PROGRAM P1_Camera
VAR
		stPos					:ST_PosData;
		tCycleTime				:TON;
		i						:INT;
		tPalletStartTime		:TON;
		nCycle_Idx				:BYTE;
		arrMES_Temp				:ARRAY [0..2] OF ST_P1MesData;
END_VAR

(*Időzítők***************************************************)
IF (stPos.nState>10000) AND (stPos.nState<100000) AND NOT tCycleTime.Q THEN
	stPos.nCycleTime := TIME_TO_REAL(tCycleTime.ET)/1000;
END_IF
tCycleTime(IN:= (stPos.nState>10000) AND (stPos.nState<150000), PT:= T#200S);							// A palettára várakozás nincs beszámolva
tPalletStartTime(IN:= NOT i_bP2PalletSensor AND fbConveyor_1.bMotorOn, PT:= T#4S);					// Alaphelyzet felvétel késleltetése!

(*Triggerek**************************************************)

(*Vész rendszer**********************************************)
IF	(NOT (i_bEmyOK AND fbDoor.bDoorsLocked) AND stPos.nState > 0) OR									// Nincs vészkör, vagy
	(NOT i_bDoorOK AND (stPos.nState>=60 AND stPos.nState<=1000)) OR									// alaphelyzetfelvétel közbe megszűnik az ajtókör vagy
	(NOT i_bDoorOK AND (stPos.nState>=10060 AND stPos.nState<=100060)) THEN							// folyamat közbe megszűnik az ajtókör 
		stPos.nState := 0;
END_IF;

(*Hibakezelés************************************************)
IF stPos.nState > 0 AND stPos.nState < 150000 THEN
	stPos.nStateLast := stPos.nState;
	IF	fbP1Lift.bError OR
		fbP1PalletDataExchange.bError OR
		(fbP1AxisX.bError AND i_bDoorOK (*AND stP1.nState >= 500*)) OR
		(fbP1AxisY.bError AND i_bDoorOK (*AND stP1.nState >= 500*)) OR
		(fbP1AxisZ.bError AND i_bDoorOK (*AND stP1.nState >= 500*)) OR
		stPos.bError THEN
			stPos.nState := 200000;
	END_IF
END_IF

(*Engedélyek *************************************************)
IF stPos.nState <= 10000
	OR stPos.nState = 100000
	OR stPos.nState = 150000
	OR stPos.nState >= 200000
THEN
	stPos.bManualModeEnable := TRUE;
ELSE
	stPos.bManualModeEnable := FALSE;
END_IF

IF stPos.nState = 0
	OR stPos.nState = 10000
	OR stPos.nState = 100000
	OR stPos.nState = 150000
	OR stPos.nState >= 200000
THEN
	stPos.bDoorOpenEnable := TRUE;
ELSE
	stPos.bDoorOpenEnable := FALSE;
END_IF

(*Kézi üzem *************************************************)
IF bManualMode THEN
	stPos.nState := 150000;
END_IF

(*Automata üzem *********************************************)
CASE stPos.nState OF
{region "Init process"}
	0:		stPos.sState := CONCAT(UDINT_TO_STRING(stPos.nState) ,' - Vészkör vagy ajtókör bontva - Működtetések törlése');
			fbP1AxisX.bGoPosition := FALSE;
			fbP1AxisY.bGoPosition := FALSE;
			fbP1AxisZ.bGoPosition := FALSE;
			fbP1Lift.bBasePosCmd := TRUE;
			fbP1Lift.bWorkPosCmd := FALSE;
			fbP1PalletDataExchange.eCommand := NoCmd;
			stPos.bError := FALSE;
			stPos.nErrorCode := 0;
			IF i_bDoorOK THEN
				IF bStepEnable THEN
					stPos.nState := stPos.nState + 20;
				END_IF
			END_IF
			
	20:		stPos.sState := CONCAT(UDINT_TO_STRING(stPos.nState) ,' - Alaphelyzetfelvétel - Kiemelő alaphelyzetbe');
			fbP1Lift.bBasePosCmd := TRUE;
			fbP1Lift.bWorkPosCmd := FALSE;
			IF fbP1Lift.bBasePosStab THEN
				IF bStepEnable THEN
					stPos.nState := stPos.nState + 20;
				END_IF
			END_IF
			
	40:		stPos.sState := CONCAT(UDINT_TO_STRING(stPos.nState) ,' - AX5805 safety ellenőrzés');	
			IF (i_bAX5805ErrorX OR i_bAX5805ErrorX) AND NOT q_bAX5805_Ack THEN
				q_bAX5805_Ack := TRUE;
			ELSIF NOT (i_bAX5805ErrorX OR i_bAX5805ErrorY OR i_bAX5805ErrorZ) THEN
				q_bAX5805_Ack := FALSE;
				IF bStepEnable THEN
					stPos.nState := stPos.nState + 20;
				END_IF
			END_IF

	60:		stPos.sState := CONCAT(UDINT_TO_STRING(stPos.nState) ,' - Szervo X tengely drive ellenőrzés');	
			IF NOT fbP1AxisX.Axis.Status.DriveDeviceError THEN
				IF bStepEnable THEN
					stPos.nState := stPos.nState + 20;
				END_IF
			END_IF

	80:		stPos.sState := CONCAT(UDINT_TO_STRING(stPos.nState) ,' - Szervo X tengely NC ellenőrzés');	
			IF NOT fbP1AxisX.Axis.Status.Error THEN
				IF bStepEnable THEN
					stPos.nState := stPos.nState + 20;
				END_IF
			END_IF

	100:	stPos.sState := CONCAT(UDINT_TO_STRING(stPos.nState) ,' - Szervo X tengely ellenőrzés');	
			IF fbP1AxisX.nState = 1000 THEN
				IF bStepEnable THEN
					stPos.nState := stPos.nState + 20;
				END_IF
			END_IF
			
	120:	stPos.sState := CONCAT(UDINT_TO_STRING(stPos.nState) ,' - Szervo Y tengely drive ellenőrzés');	
			IF NOT fbP1AxisY.Axis.Status.DriveDeviceError THEN
				IF bStepEnable THEN
					stPos.nState := stPos.nState + 20;
				END_IF
			END_IF

	140:	stPos.sState := CONCAT(UDINT_TO_STRING(stPos.nState) ,' - Szervo Y tengely NC ellenőrzés');	
			IF NOT fbP1AxisY.Axis.Status.Error THEN
				IF bStepEnable THEN
					stPos.nState := stPos.nState + 20;
				END_IF
			END_IF

	160:	stPos.sState := CONCAT(UDINT_TO_STRING(stPos.nState) ,' - Szervo Y tengely ellenőrzés');	
			IF fbP1AxisY.nState = 1000 THEN
				IF bStepEnable THEN
					stPos.nState := stPos.nState + 20;
				END_IF
			END_IF

	180:	stPos.sState := CONCAT(UDINT_TO_STRING(stPos.nState) ,' - Szervo Z tengely drive ellenőrzés');	
			IF NOT fbP1AxisZ.Axis.Status.DriveDeviceError THEN
				IF bStepEnable THEN
					stPos.nState := stPos.nState + 20;
				END_IF
			END_IF

	200:	stPos.sState := CONCAT(UDINT_TO_STRING(stPos.nState) ,' - Szervo Z tengely NC ellenőrzés');	
			IF NOT fbP1AxisZ.Axis.Status.Error THEN
				IF bStepEnable THEN
					stPos.nState := stPos.nState + 20;
				END_IF
			END_IF

	220:	stPos.sState := CONCAT(UDINT_TO_STRING(stPos.nState) ,' - Szervo Z tengely ellenőrzés');	
			IF fbP1AxisZ.nState = 1000 THEN
				IF bStepEnable THEN
					stPos.nState := 500;
				END_IF
			END_IF
	 
			
	500:	stPos.sState := CONCAT(UDINT_TO_STRING(stPos.nState) ,' - Z tengely alaphelyzetbe mozgatása');			
			fbP1AxisZ.rPosition1 := 0;
			fbP1AxisZ.rVelocity1 := 100;
			fbP1AxisZ.bGoPosition := TRUE;
			IF fbP1AxisZ.bDone THEN
				IF bStepEnable THEN
					fbP1AxisZ.bGoPosition := FALSE;
					stPos.nState := stPos.nState + 20;
				END_IF
			END_IF
			
	520:	stPos.sState := CONCAT(UDINT_TO_STRING(stPos.nState) ,' - X tengely alaphelyzetbe mozgatása');			
			fbP1AxisX.rPosition1 := 0;
			fbP1AxisX.rVelocity1 := 100;
			fbP1AxisX.bGoPosition := TRUE;
			IF fbP1AxisX.bDone THEN
				IF bStepEnable THEN
					fbP1AxisX.bGoPosition := FALSE;
					stPos.nState := stPos.nState + 20;
				END_IF
			END_IF
			
	540:	stPos.sState := CONCAT(UDINT_TO_STRING(stPos.nState) ,' - Y tengely alaphelyzetbe mozgatása');			
			fbP1AxisY.rPosition1 := 0;
			fbP1AxisY.rVelocity1 := 100;
			fbP1AxisY.bGoPosition := TRUE;
			IF fbP1AxisY.bDone THEN
				IF bStepEnable THEN
					fbP1AxisY.bGoPosition := FALSE;
					stPos.nState := stPos.nState + 20;
				END_IF
			END_IF
					 
	560:	stPos.sState := CONCAT(UDINT_TO_STRING(stPos.nState) ,' - Várakozás paletta mozgásra a pzíciók között');
			IF tPalletStartTime.Q THEN									// Normál esetben nem kerülhet ebbe az állapotba a berendezés!
				IF bStepEnable THEN										// Ha viszont P1 elengedi a palettát, amin jó termék van, és az még nem érkezik meg P2-be
					stPos.nState := 10000;								// a következő paletta ami üres megérkezik P1-be, ekkor nyomnak egy vészstopot, kinyitják az ajtót és visszahúzzák
				END_IF													// a palettát P2 elől, akkor induláskor P1 rögtön elengedné az üres palettát igy P2-be 2 paletta érkezne!!!!
			END_IF														// Ebből a hibából automatikusan csak selejtezéssel lehetne kiszedni az állomást!!! Ez nem lenne túl szerencsés!!

{endregion}
			
(* Alaphelyzet *********************************************************************)
	10000:	stPos.sState := CONCAT(UDINT_TO_STRING(stPos.nState) ,' - Alaphelyzet, termékre vár');
			IF fbP1RFID.bTagPresent AND fbP1Stopper.bPalletAtStopper AND NOT bP1ScrapRepeatError THEN
				IF bStepEnable THEN
					stPos.nState := stPos.nState + 20;
				END_IF
			END_IF	

{region "Pallet receive"}
	(*-----=== Hordozólap adatok lekérdezése ST10-től ===-----*)
	10020:	stPos.sState := CONCAT(UDINT_TO_STRING(stPos.nState) ,' - Paletta adatok lekérdezése');
			fbP1PalletDataExchange.nIndex := fbP1RFID.nTAGData;
			IF bStepEnable THEN
				fbP1PalletDataExchange.eCommand := Read;
				stPos.nState := stPos.nState + 20;
			END_IF
			
	(*-----=== Hordozólap adatok lekérdezése ST10-től ===-----*)
	10040:	stPos.sState := CONCAT(UDINT_TO_STRING(stPos.nState) ,' - Paletta adatok lekérdezése');
			IF fbP1PalletDataExchange.bDone AND NOT fbP1PalletDataExchange.bError THEN
				IF bStepEnable THEN
					fbP1PalletDataExchange.eCommand := NoCmd;
					stPos.nState := stPos.nState + 20;
				END_IF
			END_IF

	(*-----=== Hordozólap adatok kiértékelése ===-----*)
	10060:	stPos.sState := CONCAT(UDINT_TO_STRING(stPos.nState) ,' - Paletta adatok lekérdezése');
			IF		stP1PalletData.nPalletState = 2 AND			// OK termék a palettán
					stP1PalletData.nDone.3 AND					// Diszpenzálás kész
					NOT stP1PalletData.nDone.4 THEN				// Kamerás ell. még nincs kész
						IF bStepEnable THEN						// Mehet a kiemelés -> Normál folyamat
							nCycle_Idx := 0;

							arrMES_Temp[0].nOP_Index := nP1GapFillerCheckCover_Index;
							arrMES_Temp[0].sDMC_Code := stP1PalletData.sCoverCode;
							arrMES_Temp[0].sOP_Name := 'OP_GAP_FILLER_CHK_COVER';
							
							arrMES_Temp[1].nOP_Index := nP1CheckSim_Index;
							arrMES_Temp[1].sDMC_Code := stP1PalletData.sMRTCode;
							arrMES_Temp[1].sOP_Name := 'OP_CHECK_SIM';
	
							arrMES_Temp[2].nOP_Index := nP1CheckComponent_Index;
							arrMES_Temp[2].sDMC_Code := stP1PalletData.sMRTCode;
							arrMES_Temp[2].sOP_Name := 'OP_CHECK_COMPONENT';
	
							stPos.nState := stPos.nState + 20;
						END_IF
			ELSIF	stP1PalletData.nPalletState = 41 THEN		// Teszt hordozólap a kamerához
						IF bStepEnable THEN						// Még nincs funkció -> Tovább engedés
							stPos.nState := 96060; //????
						END_IF
			ELSIF	stP1PalletData.nPalletState = 2 AND			// OK termék a palettán
					NOT stP1PalletData.nDone.3 THEN				// Diszpenzálás nincs kész !
						IF bStepEnable THEN						// Átemelt hordozólap!?!? -> Selejtezés
							stP1PalletData.nPalletState := 1;
							stP1PalletData.nDone.4	:= TRUE;
							stP1PalletData.nErrorCode := 4100;
							stPos.nState := 96000;
						END_IF
			ELSIF	stP1PalletData.nPalletState = 1 THEN		// Selejt termék a palettán
						IF bStepEnable THEN						// Nincs kiemelés -> Tovább engedés
							stPos.nState := 96060;
						END_IF
			ELSIF	stP1PalletData.nPalletState = 0 THEN		// Üres paletta
						IF bStepEnable THEN						// Nincs kiemelés -> Tovább engedés
							stPos.nState := 96060;
						END_IF
			ELSE												// Nincs teendő, más állomásnak szánt hordozólap
						IF bStepEnable THEN						// Nincs kiemelés -> Tovább engedés
							stPos.nState := 96060;
						END_IF			
			END_IF

	(*-----=== MES engedély ellenőrzése ===-----*)
	10080:	stPos.sState := CONCAT(UDINT_TO_STRING(stPos.nState) ,' - MES engedély ellenőrzése');
			IF bMesEnable THEN
				IF bStepEnable THEN
					stPos.nState := 14000;
				END_IF
			ELSE
				IF bStepEnable THEN
					stPos.nState := 16000;
				END_IF				
			END_IF
{endregion}

{region "Normal process"} 
(*-----=== Recept lista kezelés ===-----*)
(* Get MRT OP state *)
14000:		stPos.sState := CONCAT(UDINT_TO_STRING(stPos.nState) ,' - Get OP state MRT (1026)');
			IF fbP1MesInterface.GET_CURRENT_OPERATION_STATE(stP1PalletData.sMRTCode, 0,stP1MesOpState) THEN
				IF stP1MesResp.RESP_CODE = '0' or stP1MesResp.RESP_CODE = '377'	THEN									// MRT OP state OK
					IF bStepEnable THEN
						stP1MrtMaterial.MATERIAL := stP1MesOpState.MAT_NO;
						stP1MrtMaterial.REVISION := stP1MesOpState.REVISION;
						nCycle_Idx := 0;
						stPos.nState := 14100;
					END_IF		
				ELSE
					IF bStepEnable THEN													// Get OP state hiba
						stP1PalletData.nPalletState := 1;
						stP1PalletData.nDone.4	:= TRUE;
							stP1PalletData.nErrorCode := 4101;
						stPos.nState := 96000;
					END_IF
				END_IF
			END_IF

	 
14100:		stPos.sState := CONCAT(UDINT_TO_STRING(stPos.nState) ,' - Get Material Custom Data (1037)');
			IF fbP1MesInterface.GET_MAT_CUSTOM_DATA(stP1MrtMaterial, 0) THEN
				IF stP1MesResp.RESP_CODE = '0'	THEN									// Get Custom Data OK
					IF bStepEnable THEN
						stPos.nState := stPos.nState + 20;
					END_IF		
				ELSE
					IF bStepEnable THEN													// Get Custom Data hiba
						stP1PalletData.nPalletState := 1;
						stP1PalletData.nDone.4	:= TRUE;
							stP1PalletData.nErrorCode := (4102 + nCycle_Idx);
						stPos.nState := 96000;
					END_IF
				END_IF
			END_IF		  

14120:		stPos.sState := CONCAT(UDINT_TO_STRING(stPos.nState) ,' - Get Custom Data By Key');
			IF fbP1MesInterface.GET_CUSTOM_DATA_BY_KEY(CONCAT(arrMES_Temp[nCycle_Idx].sOP_Name, '_R'), arrMES_Temp[nCycle_Idx].sOP_CustomData) THEN
				IF arrMES_Temp[nCycle_Idx].sOP_CustomData <> ''	THEN					// Get Custom Data by key OK
					IF bStepEnable THEN
						arrMES_Temp[nCycle_Idx].sOP_ReceipeList := arrMES_Temp[nCycle_Idx].sOP_CustomData;
						stPos.nState := stPos.nState + 20;
					END_IF		
				ELSE
					IF bStepEnable THEN													// Get Custom Data by key hiba
						stP1PalletData.nPalletState := 1;
						stP1PalletData.nDone.4	:= TRUE;
							stP1PalletData.nErrorCode := (4103 + nCycle_Idx);
						stPos.nState := 96000;
					END_IF
				END_IF
			END_IF		  

14140:		stPos.sState := CONCAT(UDINT_TO_STRING(stPos.nState) ,' - Recept lista ellenőrzése');   
			IF nCycle_Idx >= 2 THEN
				IF bStepEnable THEN						// Custom fied-ek átemelve -> Gyí, gyí gyí !!!
					nCycle_Idx := 0;
					stPos.nState := 14200;
				END_IF
			ELSE
				IF bStepEnable THEN
					nCycle_Idx := nCycle_Idx + 1;		// Van még háta Custom fiel -> Mehet a köv. lekérdezés
					stPos.nState := 14100;
				END_IF
			END_IF		

14200:
			stPos.nState := 15000;		

				 
(*-----=== MES 3010 (Start SFC) ===-----*)
	15000:	stPos.sState := CONCAT(UDINT_TO_STRING(stPos.nState) ,' - Start SFC (3010)');
			eP1GapFillerCheck_Result := E_TEST_STATE.PASSED;	
			IF fbP1MesInterface.START_SFC(arrMES_Temp[nCycle_Idx].sDMC_Code, arrMES_Temp[nCycle_Idx].nOP_Index) THEN
				IF stP1MesResp.RESP_CODE = '0'	THEN									// Jó termék
					IF bStepEnable THEN
						stPos.nState := stPos.nState + 20;
					END_IF		
				ELSE
					IF bStepEnable THEN													// Selejt
						stP1PalletData.nPalletState := 1;
						stP1PalletData.nDone.4	:= TRUE;
							stP1PalletData.nErrorCode := 4111 + nCycle_Idx;
						stPos.nState := 96000;
					END_IF
				END_IF
			END_IF

(*			// Custom field olvasása miatt kiesik! A receptlistát előre le kell tölteni! 2021.02.15
	15020:	stP1.sState := CONCAT(UDINT_TO_STRING(stP1.nState) ,' - Get recipe name');	
			IF fbP1MesInterface.GET_RECIPE_NAME_BY_OPERATION_JSON(arrMES_Temp[nCycle_Idx].sOP_Name, sP1RecipeName) THEN
			IF sP1RecipeName <>'' THEN
				stP1.nState := 16000;
			ELSE
				stP1PalletData.nPalletState := 1;							// Nincs recept név, viszont az SFC startolva -> le kell zárni hibával.
				stP1PalletData.nDone.4	:= TRUE;
				stP1PalletData.nErrorCode := 4103;
				eP1GapFillerCheck_Result := E_TEST_STATE.FAILED;
				stP1NcDat.MESDAT[stP1NcDat.N].RESPONSE_CODE := '4103';
				stP1NcDat.MESDAT[stP1NcDat.N].RESPONSE_DESCRIPTION := CONCAT(CONCAT('The ',arrMES_Temp[nCycle_Idx].sOP_Name),' recipe missing');
				stP1NcDat.MESDAT[stP1NcDat.N].CLIENT_DATE := fbP1MesInterface.GET_LOCAL_TIME();
				stP1NcDat.MESDAT[stP1NcDat.N].TEST_STATE := INT_TO_STRING(E_TEST_STATE.FAILED);
				stP1NcDat.MESDAT[stP1NcDat.N].TEST_STEP := INT_TO_STRING(stP1NcDat.N);
				stP1NcDat.MESDAT[stP1NcDat.N].VALUE := '0';
				stP1.nState := 95000;
			END_IF
		END_IF
*)

	15020:	stPos.sState := CONCAT(UDINT_TO_STRING(stPos.nState) ,' - Receptnév átadása');	
			fbP1ReceipeList(
				sReceipeListIn:= arrMES_Temp[nCycle_Idx].sOP_ReceipeList,
				sReceipeListOut=> arrMES_Temp[nCycle_Idx].sOP_ReceipeList,
				sReceipe=> sP1RecipeName,
				bEmpty=> );
			stPos.nState := 16000;

(*-----=== Recept kezelés ===-----*)
	16000:	stPos.sState := CONCAT(UDINT_TO_STRING(stPos.nState) ,' - Recept lista frissítése');
			bP1RecipeRefresh := TRUE;
			IF fbP1RecipeManager.DONE AND fbP1RecipeManager.RECIPE_CNT > 0 THEN
				IF bStepEnable THEN
						bP1RecipeRefresh := FALSE;
						stPos.nState := stPos.nState + 20;
				END_IF
			END_IF

	16020:	stPos.sState := CONCAT(UDINT_TO_STRING(stPos.nState) ,' - Várakozás recept lista frissítés befejezésére');
			IF NOT fbP1RecipeManager.DONE AND NOT fbP1RecipeManager.RESET THEN
				IF bMesEnable THEN
					IF bStepEnable THEN
							stPos.nState := stPos.nState + 20;
					END_IF
				ELSE
					IF bStepEnable THEN
							sP1RecipeName := arrP1RecipeNames[nCycle_Idx + 1];			// Kikapcsolt MES esetén is legyen ellenőrzés 
							stPos.nState := stPos.nState + 20;
					END_IF
				END_IF
			END_IF

	16040:	stPos.sState := CONCAT(UDINT_TO_STRING(stPos.nState) ,' - Recept betöltése');
			bP1RecipeLoad := TRUE;
			IF fbP1RecipeManager.DONE THEN
				IF bStepEnable THEN
						bP1RecipeLoad := FALSE;
						i := 0;
						stP1NcDat.N := 1;
						stPos.nState := stPos.nState + 20;
				END_IF
			END_IF

	16060:	stPos.sState := CONCAT(UDINT_TO_STRING(stPos.nState) ,' - Várakozás recept betöltés befejezésére');
			IF NOT fbP1RecipeManager.DONE AND NOT fbP1RecipeManager.RESET THEN
				IF NOT fbP1RecipeManager.READ_FILE.ERROR THEN
					IF bStepEnable THEN
							stPos.nState := stPos.nState + 20;			// Recept betöltés kész
					END_IF
				ELSE
					stP1PalletData.nPalletState := 1;					// Nincs recept név, viszont az SFC startolva -> le kell zárni hibával.
					stP1PalletData.nDone.4	:= TRUE;
					stP1PalletData.nErrorCode := 4104;
					eP1GapFillerCheck_Result := E_TEST_STATE.FAILED;
					stP1NcDat.MESDAT[stP1NcDat.N].RESPONSE_CODE := '4113';
					stP1NcDat.MESDAT[stP1NcDat.N].RESPONSE_DESCRIPTION := CONCAT(CONCAT('The ',arrMES_Temp[nCycle_Idx].sOP_Name),' recipe not found');
					stP1NcDat.MESDAT[stP1NcDat.N].CLIENT_DATE := fbP1MesInterface.GET_LOCAL_TIME();
					stP1NcDat.MESDAT[stP1NcDat.N].TEST_STATE := INT_TO_STRING(E_TEST_STATE.FAILED);
					stP1NcDat.MESDAT[stP1NcDat.N].TEST_STEP := INT_TO_STRING(stP1NcDat.N);
					stP1NcDat.MESDAT[stP1NcDat.N].VALUE := '0';
					stPos.nState := 95000;
				END_IF
			END_IF

	16080:	stPos.nState := 18000;


(*-----=== Normál folyamat ===-----*)
	18000:	stPos.sState := CONCAT(UDINT_TO_STRING(stPos.nState) ,' - Kiemelő munkahelyzetbe');
			fbP1Lift.bBasePosCmd := FALSE;
			fbP1Lift.bWorkPosCmd := TRUE;
			IF fbP1Lift.bWorkPosStab THEN
				IF bStepEnable THEN
					stPos.nState := stPos.nState + 20;
				END_IF
			END_IF

	18020:	stPos.sState := CONCAT(UDINT_TO_STRING(stPos.nState) ,' - Programlépés betöltése');
			fbP1AxisX.rPosition1 := LREAL_TO_REAL(stP1Recipe.Seq[i].Target.X);
			fbP1AxisX.rVelocity1 := rVelocity;
			fbP1AxisY.rPosition1 := LREAL_TO_REAL(stP1Recipe.Seq[i].Target.Y);
			fbP1AxisY.rVelocity1 := rVelocity;
			fbP1AxisZ.rPosition1 := LREAL_TO_REAL(stP1Recipe.Seq[i].Target.Z);
			fbP1AxisZ.rVelocity1 := rVelocity;
			fbP1Cam1.nProgNr := INT_TO_UINT(stP1Recipe.Seq[i].CheckingProgramId);
			IF bStepEnable THEN
					stPos.nState := stPos.nState + 20;
			END_IF
			
	18040:	stPos.sState := CONCAT(UDINT_TO_STRING(stPos.nState) ,' - X,Y,Z tengely pozícióba mozgatása');						
			fbP1AxisX.bGoPosition := TRUE;
			fbP1AxisY.bGoPosition := TRUE;
			fbP1AxisZ.bGoPosition := TRUE;
			IF fbP1AxisX.bDone AND fbP1AxisY.bDone AND fbP1AxisZ.bDone THEN
				IF bStepEnable THEN
					fbP1AxisX.bGoPosition := FALSE;
					fbP1AxisY.bGoPosition := FALSE;
					fbP1AxisZ.bGoPosition := FALSE;
					stPos.nState := stPos.nState + 20;
				END_IF
			END_IF
			
	18060:	stPos.sState := CONCAT(UDINT_TO_STRING(stPos.nState) ,' - Kamera triggerelése');						
			fbP1Cam1.bStart := TRUE;
			IF NOT fbP1Cam1.bReady AND NOT fbP1Cam1.bBusy THEN			
				IF bStepEnable THEN
					stPos.nState := stPos.nState + 20;
				END_IF
			END_IF
			
	18080:	stPos.sState := CONCAT(UDINT_TO_STRING(stPos.nState) ,' - Kiértékelés');						
			IF	fbP1Cam1.bFail THEN
					fbP1Cam1.bStart := FALSE;
					nP1ScrapCounter := nP1ScrapCounter + 1;
					stP1PalletData.nPalletState := 1;								// Fail -> Hordozólap selejt
					stP1PalletData.nDone.4	:= TRUE;
					stP1PalletData.nErrorCode := INT_TO_WORD(4121 + i);
					eP1GapFillerCheck_Result := E_TEST_STATE.FAILED;
					stP1NcDat.MESDAT[stP1NcDat.N].RESPONSE_CODE := INT_TO_STRING(4121 + i);
					stP1NcDat.MESDAT[stP1NcDat.N].RESPONSE_DESCRIPTION := CONCAT('Camera error of POS#', INT_TO_STRING(i));
					stP1NcDat.MESDAT[stP1NcDat.N].CLIENT_DATE := fbP1MesInterface.GET_LOCAL_TIME();
					stP1NcDat.MESDAT[stP1NcDat.N].TEST_STATE := INT_TO_STRING(E_TEST_STATE.FAILED);
					stP1NcDat.MESDAT[stP1NcDat.N].TEST_STEP := INT_TO_STRING(stP1NcDat.N);
					stP1NcDat.MESDAT[stP1NcDat.N].VALUE := '0';
					stPos.nState := 95000;	
			ELSE
				fbP1Cam1.bStart := FALSE;
				stPos.nState := stPos.nState + 20;
			END_IF

	18100:	stPos.sState := CONCAT(UDINT_TO_STRING(stPos.nState) ,' - Recept kész?');
			IF	stP1Recipe.Seq[i].LastPosition THEN
					IF fbP1ReceipeList.bEmpty THEN
						stPos.nState := 95000;							// A recept kész és ez volt az utolsó a listába
					ELSE
						stPos.nState := 15020;							// A recept kész de nem ez volt az utolsó a listába! -> Új recept betöltése!
					END_IF
			ELSE 
				i := i+1;												// A recept még nincs kész
				stPos.nState := 18020;
			END_IF
	
(*-----=== MES 3503 (Log NC Data) ===-----*)
	95000:	stPos.sState := CONCAT(UDINT_TO_STRING(stPos.nState) ,' - Log NC (3503)');	
			IF stP1PalletData.nPalletState = 1 AND bMesEnable THEN
				IF fbP1MesInterface.ASSY_SAVE_NCDAT(arrMES_Temp[nCycle_Idx].sDMC_Code,arrMES_Temp[nCycle_Idx].nOP_Index,stP1NcDat) THEN
					IF bStepEnable THEN
						stPos.nState := stPos.nState + 20;			// A paletta már selejt és van bent hibakód! Nincs felülírás.
					END_IF							
				END_IF
			ELSE
				IF bStepEnable THEN
					stPos.nState := stPos.nState + 20;
				END_IF
			END_IF

(*-----=== MES 3011 (Complete SFC) ===-----*)
	95020:	stPos.sState := CONCAT(UDINT_TO_STRING(stPos.nState) ,' - Complete SFC (3011)');
			IF bMesEnable THEN	
				IF fbP1MesInterface.COMPLETE_SFC(arrMES_Temp[nCycle_Idx].sDMC_Code, arrMES_Temp[nCycle_Idx].nOP_Index, eP1GapFillerCheck_Result) THEN
					IF stP1MesResp.RESP_CODE='0' THEN
						stPos.nState := stPos.nState + 20;
					ELSE
						stP1PalletData.nPalletState := 1;			// A MES-be aktív marad nem tudom selejtezni! Csak a hordozót selejtezem
						stP1PalletData.nErrorCode := 4114;
						stPos.nState := stPos.nState + 20;
					END_IF
				END_IF
			ELSE
				stPos.nState := stPos.nState + 20;
			END_IF


	95040:	stPos.sState := CONCAT(UDINT_TO_STRING(stPos.nState) ,' - Folyamat ellenőrzése');
			IF stP1PalletData.nPalletState = 1 OR nCycle_Idx >= 2 THEN
				IF bStepEnable THEN						// Selejt vagy kész a folyamat -> Lejelentés
					stP1PalletData.nDone.4 := TRUE;
					stPos.nState := stPos.nState + 20;
				END_IF
			ELSE
				IF bStepEnable THEN
					nCycle_Idx := nCycle_Idx + 1;		// Jó termék és még nincs kész a folyamat -> Mehet a köv. folyamat
					IF bMesEnable THEN
						stPos.nState := 15000;
					ELSE
						stPos.nState := 16000;
					END_IF
				END_IF
			END_IF
			
	95060:		
			stPos.nState := 96000;

	(*-----=== Hordozólap adatok feltöltése ST10-be ===-----*)
	96000:	stPos.sState := CONCAT(UDINT_TO_STRING(stPos.nState) ,' - Paletta adatok feltöltése');
			fbP1PalletDataExchange.nIndex := fbP1RFID.nTAGData;
			IF bStepEnable THEN
				fbP1PalletDataExchange.eCommand := Write;
				stPos.nState := stPos.nState + 20;
			END_IF
			
	(*-----=== Hordozólap adatok feltöltése ST10-be ===-----*)
	96020:	stPos.sState := CONCAT(UDINT_TO_STRING(stPos.nState) ,' - Paletta adatok feltöltése');
			IF fbP1PalletDataExchange.bDone AND NOT fbP1PalletDataExchange.bError THEN
				IF bStepEnable THEN
					fbP1PalletDataExchange.eCommand := NoCmd;
					stPos.nState := stPos.nState + 20;
				END_IF
			END_IF

	96040:	stPos.sState := CONCAT(UDINT_TO_STRING(stPos.nState) ,' - X,Y tengely pozícióba mozgatása');
			fbP1AxisX.rPosition1 := 0;
			fbP1AxisX.rVelocity1 := rVelocity;
			fbP1AxisY.rPosition1 := 0;
			fbP1AxisY.rVelocity1 := rVelocity;					
			fbP1AxisZ.rPosition1 := 0;
			fbP1AxisZ.rVelocity1 := rVelocity;					
			fbP1AxisX.bGoPosition := TRUE;
			fbP1AxisY.bGoPosition := TRUE;
			fbP1AxisZ.bGoPosition := TRUE;
			IF fbP1AxisX.bDone AND fbP1AxisY.bDone AND fbP1AxisZ.bDone THEN
				IF bStepEnable THEN
					fbP1AxisX.bGoPosition := FALSE;
					fbP1AxisY.bGoPosition := FALSE;
					fbP1AxisZ.bGoPosition := FALSE;
					stPos.nState := stPos.nState + 20;
				END_IF
			END_IF		
	
	96060:	stPos.sState := CONCAT(UDINT_TO_STRING(stPos.nState) ,' - Kiemelő alaphelyzetbe');
			fbP1Lift.bBasePosCmd := TRUE;
			fbP1Lift.bWorkPosCmd := FALSE;
			IF fbP1Lift.bBasePosStab THEN
				IF bStepEnable THEN
					i:=0;
					stPos.nState := stPos.nState + 20;	
				END_IF
			END_IF		

	96080:	stPos.sState := CONCAT(UDINT_TO_STRING(stPos.nState) ,' - Ismétlődő hibák ellenőrzése');
			IF NOT bP1ScrapRepeatError THEN
				stPos.nState := 100000;
			END_IF
{endregion}
			
(*-----=== Automata ciklus befejezése ===-----*)
	100000:	stPos.sState := CONCAT(UDINT_TO_STRING(stPos.nState) ,' - Várakozás hordozólap elengedésre');
			IF NOT fbP1Stopper.bPalletAtStopper THEN
				IF bStepEnable THEN
					i:=0;
					stPos.nState := stPos.nState + 20;
				END_IF
			END_IF		

	100020:
			stPos.nState := 10000;	
			
(* Kézi üzem *********************************************************************)
	150000:	stPos.sState := CONCAT(UDINT_TO_STRING(stPos.nState) ,' - Kézi üzem');
			IF NOT bManualMode THEN
				stPos.nState := 0;
			ELSE
				;
			END_IF
			
	(* Hibakezelés *********************************************************************)
	200000:	stPos.sState := CONCAT(UDINT_TO_STRING(stPos.nState) ,CONCAT(' - Hiba, ebből az állapotból: ' ,stPos.sState));
			fbP1PalletDataExchange.eCommand := NoCmd;
			stPos.bError := TRUE;
			stPos.nState := stPos.nState + 20;

	(* Hibakezelés *********************************************************************)
	200020:	IF bAckP THEN
				CASE stPos.nStateLast OF
					(* Alaphelyzet felvétel folyamán *)
					0..9999:	stPos.nState := 0;
				ELSE 			stPos.nState := 0;
				END_CASE
				stPos.bError := FALSE;
			END_IF
ELSE
	stPos.sState := CONCAT(UDINT_TO_STRING(stPos.nState) ,' - Nem használt állapot');
END_CASE

ACTION Camera:
fbP1Cam1(
	sName:= 'CAM1 Basler acA4600-7gc', 
	bEn:= TRUE, 
	bEHA:= TRUE, 
	bAck:= bAckP, 
	timConnection:= T#1500MS, 
	timReady:= T#1500MS, 
	timProgChange:= T#1500MS, 
	timProgRun:= T#5S, 
	stCAM_IN:= stCam1_IN,
	stComErrEvent:= TC_EVENTS.MyEvent.fbP1Cam1Com,
	stReadyErrEvent:= TC_EVENTS.MyEvent.fbP1Cam1Ready,
	stProgErrEvent:= TC_EVENTS.MyEvent.fbP1Cam1Prog,
	stRunErrEvent:= TC_EVENTS.MyEvent.fbP1Cam1Run, 
	stCAM_OUT=> stCam1_OUT);
END_ACTION

ACTION DataExchange:
fbP1PalletDataExchange(
	stPalletData:= stP1PalletData, 
	sName:= 'P1 Camera pos.', 
	bAck:= bAckP, 
	sAMSNetId:= sST10_NetId, 
	stEventEntry:= TC_EVENTS.MyEvent.fbP1PalletDataExchange);
END_ACTION

ACTION Diag:
fbP1FullCycleTime(
	bPalletSensor:= fbP1Stopper.i_bPalettSensor,
	timTimeMax:= T#200S,
	nCurrentCycleTime=> ,
	arrCycleTimes=> );
END_ACTION

ACTION MES:
fbP1MesInterface(
	HOST:= '127.0.0.1', 
	PORT:= 5500, 
	ENABLE:= TRUE, 
	RESET:= fbP1MesInterface.ERROR, 
	STX:= , 
	ETX:= , 
	RESP:= stP1MesResp, 
	TEST_ADAPTER:= '0', 
	ADAPTER_ID:= '1', 
	BUSY=> , 
	READY=> , 
	DONE=> , 
	ERROR=> , 
	ERROR_ID=> );
END_ACTION

ACTION Pneu:
fbP1Lift(
	sName:= 'Z4.4', 
	sBasePosSensor:= 'S4131', 
	sWorkPosSensor:= 'S4132', 
	bEn:= i_bDoorOK, 
	bEHA:= bGlobalEHA, 
	bDisableManualCmd:= NOT bManualMode, 
	bAck:= bAckP, 
	timBasePos:= , 
	timWorkPos:= ,
	stBasePosEvent:= TC_Events.MyEvent.fbP1LiftBPE, 
	stWorkPosEvent:= TC_Events.MyEvent.fbP1LiftWPE);
END_ACTION

ACTION Recipe:
fbP1RecipeManager(
	sDef:= 'Vision', 
	sExt:= 'tcdata', 
	sFolderPath:= 'C:\TwinCAT\Tc_Data', 
	sKey:= 'Data', 
	pData:= ADR(stP1Recipe), 
	nData:= SIZEOF(stP1Recipe), 
	RESET:= , 
	READY=> , 
	BUSY=> , 
	DONE=> , 
	ERROR=> , 
	ERROR_ID=> , 
	TIME_STAMP=> , 
	RECIPE_LIST=> arrP1RecipeNames, 
	RECIPE_CNT=> );
	
IF	bP1RecipeLoad AND
	NOT bP1RecipeSave AND
	NOT bP1RecipeRefresh AND
	NOT fbP1RecipeManager.RESET AND
	NOT fbP1RecipeManager.DONE THEN
			fbP1RecipeManager.Load(NAME:= sP1RecipeName);
END_IF

IF	NOT bP1RecipeLoad AND
	bP1RecipeSave AND
	NOT bP1RecipeRefresh AND
	NOT fbP1RecipeManager.RESET AND
	NOT fbP1RecipeManager.DONE THEN
			fbP1RecipeManager.Save(NAME:= sP1RecipeName);
END_IF

IF	NOT bP1RecipeLoad AND
	NOT bP1RecipeSave AND
	bP1RecipeRefresh AND
	NOT fbP1RecipeManager.RESET AND
	NOT fbP1RecipeManager.DONE THEN
			fbP1RecipeManager.RefreshNameList();
END_IF

IF	NOT bP1RecipeLoad AND
	NOT bP1RecipeSave AND
	NOT bP1RecipeRefresh AND
	NOT fbP1RecipeManager.RESET AND
	fbP1RecipeManager.DONE THEN
			fbP1RecipeManager.RESET := TRUE;
END_IF

IF	fbP1RecipeManager.RESET AND
	NOT fbP1RecipeManager.DONE THEN
			fbP1RecipeManager.RESET := FALSE;
END_IF
END_ACTION

ACTION RFID:
fbP1RFID(sName:= 'P1 RFID');
END_ACTION

ACTION Servo:
fbP1AxisX.lrNegLimit := 0;
fbP1AxisX.lrPosLimit := 390;
fbP1AxisX.bEnableNegative := TRUE;
fbP1AxisX.bEnablePositive := TRUE;

fbP1AxisX(
	sName:= 'Axis X', 
	bEMYOK:= i_bDoorOK AND NOT i_bAX5805ErrorX, 
	bErrorAck:= bAckP, 
	bDisableManualCmd:= NOT bManualMode, 
	bBufferedMove:= FALSE,
	rVelocityJog := 10, 
	stAxisEvent:= TC_EVENTS.MyEvent.fbP1AxisX
);

fbP1AxisY.lrNegLimit := 0;
fbP1AxisY.lrPosLimit := 290;
fbP1AxisY.bEnableNegative := TRUE;
fbP1AxisY.bEnablePositive := TRUE;

fbP1AxisY(
	sName:= 'Axis Y', 
	bEMYOK:= i_bDoorOK AND NOT i_bAX5805ErrorY, 
	bErrorAck:= bAckP, 
	bDisableManualCmd:= NOT bManualMode, 
	bBufferedMove:= FALSE, 
	rVelocityJog := 10, 
	stAxisEvent:= TC_EVENTS.MyEvent.fbP1AxisY
);

fbP1AxisZ.lrNegLimit := 0;
fbP1AxisZ.lrPosLimit := 100;
fbP1AxisZ.bEnableNegative := TRUE;
fbP1AxisZ.bEnablePositive := TRUE;

fbP1AxisZ(
	sName:= 'Axis Z', 
	bEMYOK:= i_bDoorOK AND NOT i_bAX5805ErrorZ, 
	bErrorAck:= bAckP, 
	bDisableManualCmd:= NOT bManualMode, 
	bBufferedMove:= FALSE, 
	rVelocityJog := 10, 
	stAxisEvent:= TC_EVENTS.MyEvent.fbP1AxisZ
);
END_ACTION

END_PROGRAM

(* stored: Version 1.1.0.1, ProductVersion 3.1.4024.10
   POU P1_Camera: Id {34762149-00dc-4394-ac04-664d8169154b}, SpecialFunc None
   Action Camera: Id {1213996c-08f5-4059-aef6-e3e8cd24eabc}
   Action DataExchange: Id {7bde8b84-684d-4fde-adc4-5477fe0f4bf1}
   Action Diag: Id {af734140-f890-40ad-9f47-5144bf63b61b}
   Action MES: Id {9fb22461-eca9-41fe-8bdd-472edb2f70f5}
   Action Pneu: Id {f07977e9-c232-4786-bdab-dc615701d97a}
   Action Recipe: Id {a8df4282-a7c8-4c21-9b23-afeed744d1aa}
   Action RFID: Id {eaabd472-e0b4-47cd-bef9-9d6e2760fe70}
   Action Servo: Id {dcbbb598-b6a2-44d3-9d13-7dbfb1fcdc76} *)
